{attribute 'pack_mode' := '1'}
    {attribute 'OPC.UA.DA' := '1'}
    {attribute 'OPC.UA.DA.StructuredType' := '1'}
    (*
    ST_RWTime_HMI_IgnitionExp
    ==================================================
    Generated from Ignition UDT: RW_Time
    Total tags: 1
    Generated on: 2025-09-15 12:56:43
    *)
    TYPE ST_RWTime_HMI_IgnitionExp :
    STRUCT
        {attribute 'OPC.UA.DA' := '1'}
        {attribute 'OPC.UA.DA.Description' := '{Description}'}
        // {Description}
        Value : REAL := 0.0;
    END_STRUCT
    END_TYPE

(* stored: Version 1.1.0.1
   DUT ST_RWTime_HMI_IgnitionExp: Id {cd9f8a0c-c0b6-4ca7-b0b2-9b1f99c24a2d} *)
